# EPICS StreamDevice protocol: instronArbyApp/Db/devinstron.proto
#
# The stress rig appears to occasionally "hang" for a fair amount of time.
#
# Empirically, these timeouts appear to be enough to overcome the "hang"...
#
ReadTimeout = 15000;
ReplyTimeout = 15000;
WriteTimeout = 15000;
LockTimeout = 30000;

# Fake read terminator from Arby, not actually sent by device
InTerminator = CR LF;

#
# Individual commands
#

getCurrentControlChannel {
    out "Q300";
	in "%d";
}

getWatchdogStatus {
    out "Q904";
	in "%d%*s";
}

disableWatchdog {
    # out "C904,0";
}

getControlMode {
    out "Q909";
	in "%d";
}

getStatus {
    out "Q22";
    in "%d";
}

getActuatorStatus {
    out "Q23";
	in "%d";
}

getMovementType {
    out "Q1";
	in "%d";
}

#
# Blocks of commands
#

initRoutine {
}

panicStop {
    out "C23,0";
}

setMovementType {
	out "C500,%d;C38,1";
	out "C916,0";
	out "C914,4";
	out "C916,2";
	out "C372";
}

arbRW {
    out "%(\$1.VAL)s";
    in "%39c";
}

setCurrentControlChannel {
    out "C300,%d";
}

setStepTime {
    out "C86,\$1,%f";
}

getStepTime {
    out "Q86,\$1";
    in "%f";
}

setChanWaveType {
    out "C2,\$1,%d";
}

getChanWaveType {
    out "Q2,\$1";
    in "%d";
}

getRampAmpSP {
    out "Q4,\$1";
    in "%f";
}

setRampAmpSP {
    out "C4,\$1,%f";
}

getCurrentFeedback {
    out "Q134,\$1,0";
    in "%f";
}

getChanScale {
    out "Q308,\$1";
    in "%f";
}

getStrainLength {
    out "Q340,\$1";
    in "%f";
}

setArea {
    out "C341,\$1,%f";
}

getArea {
    out "Q341,\$1";
    in "%f";
}

getType {
    out "Q307,\$1";
    in "%(\$2:TYPE:STANDARD)d,%d"
}

#
# Waveform commands
#

getWaveformStatus {
    out "Q200";
    in "%d";
}

setWaveformAbort {
    out "C200,0";
}

setWaveformStart {
    out "C200,1";
}

setWaveformStop {
    out "C200,4";
}

setWaveformAmplitude {
    out "C203,%(\$1.RVAL)d,%.10f";
}

getWaveformAmplitude {
    out "Q203,%(\$1.RVAL)d";
	in "%f";
}

setWaveformFrequency {
    out "C202,%(\$1.RVAL)d,%f";
}

getWaveformFrequency {
    out "Q202,%(\$1.RVAL)d";
	in "%f";
}

setWaveformType {
    out "C201,%(\$1.RVAL)d,%d";
}

getWaveformType {
    out "Q201,%(\$1.RVAL)d";
	in "%d";
}

setWaveformQuartOff {
    out "C212,0";
}

getQuartCountsMax {
    out "Q209";
	in "%d";
}

setQuartCountsMax {
    out "C209,%d";
}

getQuartCounts {
    out "Q210";
	in "%d";
}

setWaveformHold {
    out "C213,3";
}

setLogMaintain {
    out "C214,0";
}

setWaveformQuartArm {
    out "C212,2";
}

getWaveformQuartStatus {
    out "Q212";
	in "%d";
}
